Staubli VAL3: CmdTxtReading.pgx

program CmdTxtReading()
begin
  //  call TxtHMI()
  //
  call Txt_initData()
  call Txt_PkgInit()
  nRoateTotal=5
  while true
   // if n_sTxt<nTxtTotal and nTxtTotal>2
   if n_Roate<nRoateTotal and nTxtTotal>2
      if bTxt1==true
        call TxtReadRoom1()
      else
      endIf
      if bTxt2==true
        call TxtReadRoom2()
      else
      endIf
      if bTxt3==true
        call TxtReadRoom3()
      else
      endIf
    else
    endIf
    //    nScrPts=n_sTxt
    //    call hmi_refreshmain()
  endWhile
end
